SYSTEM DRILL_MVL (* Drill System Model+View+HMI with shared simulation clock *)
  (* Standard: 61499-1; Classification: Simulation; ApplicationDomain: Transfer Lines; Function: Drilling *)
  (* Version 0.1, 2004-10-25, JHC, Rockwell Automation, Adapted to new Load/Unload model. *)
  (* Version 0.0, 2004-09-26, JHC, Rockwell Automation *)
  DEVICE MODEL : FRAME_DEVICE
    RESOURCE CLOCK : EMB_RES
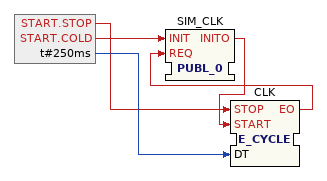
      FBS
        CLK : E_CYCLE;
        SIM_CLK : PUBL_0;
      END_FBS
      EVENT_CONNECTIONS
        START.STOP TO CLK.STOP;
        START.COLD TO SIM_CLK.INIT;
        SIM_CLK.INITO TO CLK.START;
        CLK.EO TO SIM_CLK.REQ;
      END_CONNECTIONS
      DATA_CONNECTIONS
        t#250ms TO CLK.DT;
      END_CONNECTIONS
    END_RESOURCE
    RESOURCE SUPPLY_MDL : EMB_RES
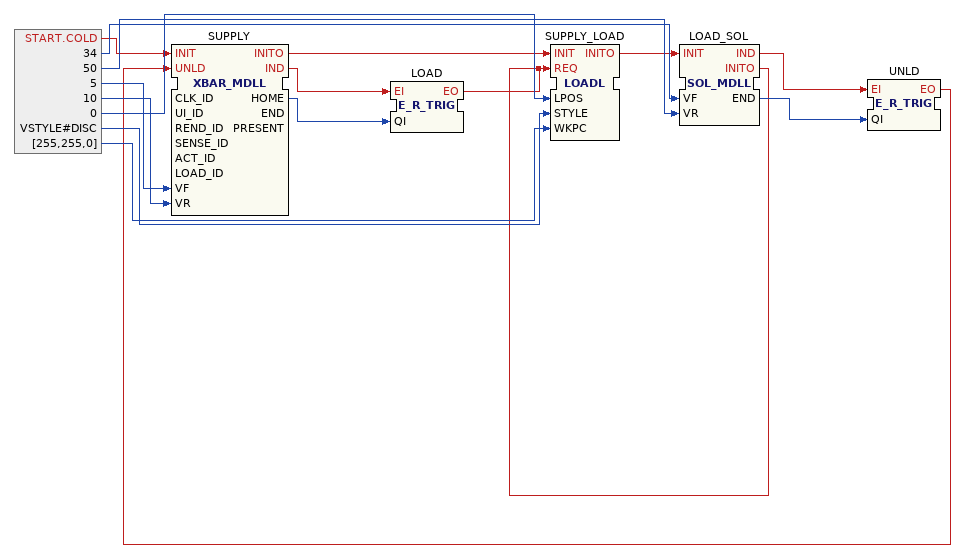
      FBS
        SUPPLY : XBAR_MDLL;
        LOAD_SOL : SOL_MDLL;
        UNLD : E_R_TRIG;
        LOAD : E_R_TRIG;
        SUPPLY_LOAD : LOADL;
      END_FBS
      EVENT_CONNECTIONS
        START.COLD TO SUPPLY.INIT;
        LOAD_SOL.IND TO UNLD.EI;
        SUPPLY.IND TO LOAD.EI;
        UNLD.EO TO SUPPLY.UNLD;
        SUPPLY.INITO TO SUPPLY_LOAD.INIT;
        SUPPLY_LOAD.INITO TO LOAD_SOL.INIT;
        LOAD_SOL.INITO TO SUPPLY_LOAD.REQ;
        LOAD.EO TO SUPPLY_LOAD.REQ;
      END_CONNECTIONS
      DATA_CONNECTIONS
        34 TO LOAD_SOL.VF;
        50 TO LOAD_SOL.VR;
        LOAD_SOL.END TO UNLD.QI;
        5 TO SUPPLY.VF;
        10 TO SUPPLY.VR;
        SUPPLY.HOME TO LOAD.QI;
        0 TO SUPPLY_LOAD.LPOS;
        VSTYLE#DISC TO SUPPLY_LOAD.STYLE;
        [255,255,0] TO SUPPLY_LOAD.WKPC;
      END_CONNECTIONS
    END_RESOURCE
    RESOURCE SLIDE_MDL : EMB_RES
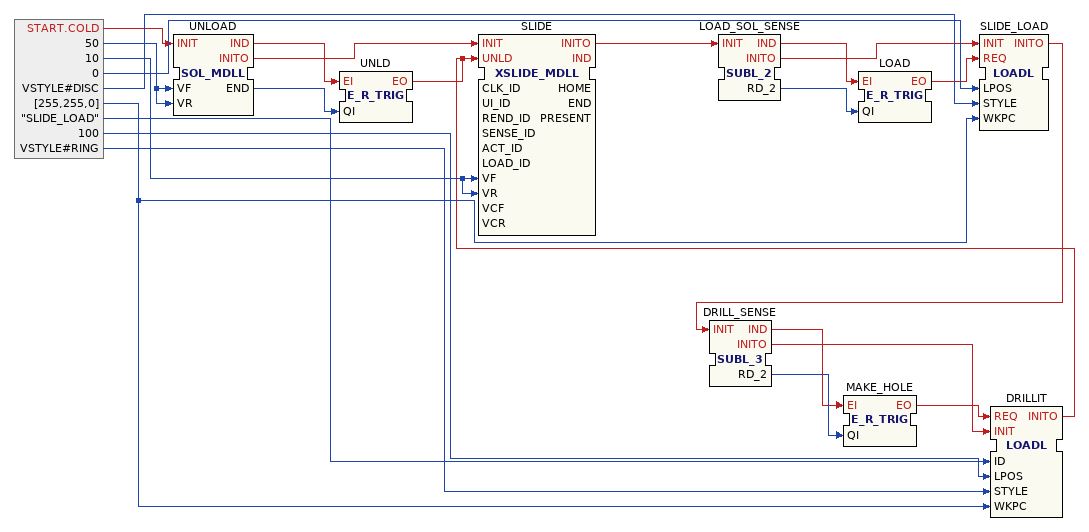
      FBS
        SLIDE : XSLIDE_MDLL;
        UNLOAD : SOL_MDLL;
        DRILL_SENSE : SUBL_3;
        MAKE_HOLE : E_R_TRIG;
        UNLD : E_R_TRIG;
        LOAD_SOL_SENSE : SUBL_2;
        LOAD : E_R_TRIG;
        SLIDE_LOAD : LOADL;
        DRILLIT : LOADL;
      END_FBS
      EVENT_CONNECTIONS
        DRILL_SENSE.IND TO MAKE_HOLE.EI;
        UNLOAD.IND TO UNLD.EI;
        UNLD.EO TO SLIDE.UNLD;
        LOAD_SOL_SENSE.IND TO LOAD.EI;
        START.COLD TO UNLOAD.INIT;
        UNLOAD.INITO TO SLIDE.INIT;
        SLIDE.INITO TO LOAD_SOL_SENSE.INIT;
        LOAD_SOL_SENSE.INITO TO SLIDE_LOAD.INIT;
        LOAD.EO TO SLIDE_LOAD.REQ;
        MAKE_HOLE.EO TO DRILLIT.REQ;
        DRILLIT.INITO TO SLIDE.UNLD;
        SLIDE_LOAD.INITO TO DRILL_SENSE.INIT;
        DRILL_SENSE.INITO TO DRILLIT.INIT;
      END_CONNECTIONS
      DATA_CONNECTIONS
        50 TO UNLOAD.VF;
        50 TO UNLOAD.VR;
        DRILL_SENSE.RD_2 TO MAKE_HOLE.QI;
        10 TO SLIDE.VF;
        10 TO SLIDE.VR;
        UNLOAD.END TO UNLD.QI;
        LOAD_SOL_SENSE.RD_2 TO LOAD.QI;
        0 TO SLIDE_LOAD.LPOS;
        VSTYLE#DISC TO SLIDE_LOAD.STYLE;
        [255,255,0] TO SLIDE_LOAD.WKPC;
        "SLIDE_LOAD" TO DRILLIT.ID;
        100 TO DRILLIT.LPOS;
        VSTYLE#RING TO DRILLIT.STYLE;
        [255,255,0] TO DRILLIT.WKPC;
      END_CONNECTIONS
    END_RESOURCE
    RESOURCE DRILL_MDL : EMB_RES
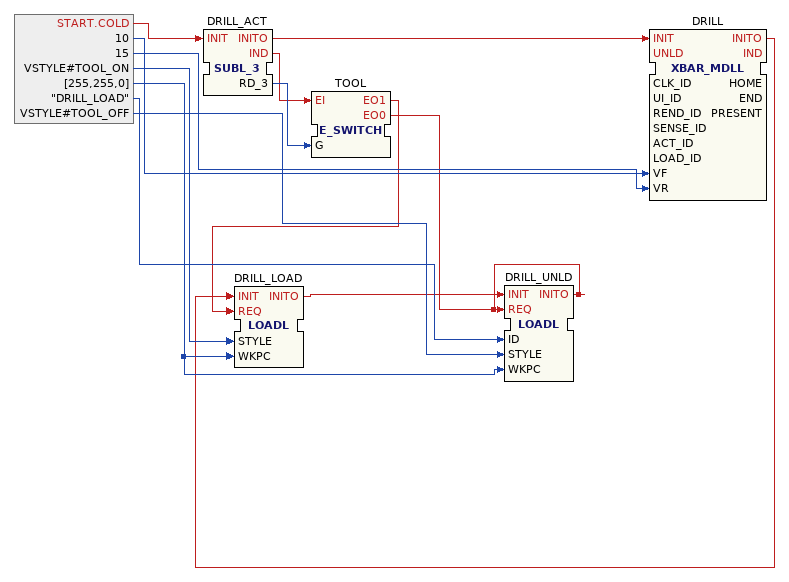
      FBS
        DRILL : XBAR_MDLL;
        DRILL_ACT : SUBL_3;
        TOOL : E_SWITCH;
        DRILL_LOAD : LOADL;
        DRILL_UNLD : LOADL;
      END_FBS
      EVENT_CONNECTIONS
        START.COLD TO DRILL_ACT.INIT;
        DRILL_ACT.INITO TO DRILL.INIT;
        DRILL.INITO TO DRILL_LOAD.INIT;
        DRILL_LOAD.INITO TO DRILL_UNLD.INIT;
        DRILL_ACT.IND TO TOOL.EI;
        TOOL.EO1 TO DRILL_LOAD.REQ;
        TOOL.EO0 TO DRILL_UNLD.REQ;
        DRILL_UNLD.INITO TO DRILL_UNLD.REQ;
      END_CONNECTIONS
      DATA_CONNECTIONS
        10 TO DRILL.VF;
        15 TO DRILL.VR;
        VSTYLE#TOOL_ON TO DRILL_LOAD.STYLE;
        [255,255,0] TO DRILL_LOAD.WKPC;
        "DRILL_LOAD" TO DRILL_UNLD.ID;
        VSTYLE#TOOL_OFF TO DRILL_UNLD.STYLE;
        [255,255,0] TO DRILL_UNLD.WKPC;
        DRILL_ACT.RD_3 TO TOOL.G;
      END_CONNECTIONS
    END_RESOURCE
    RESOURCE TAKEOFF_MDL : EMB_RES
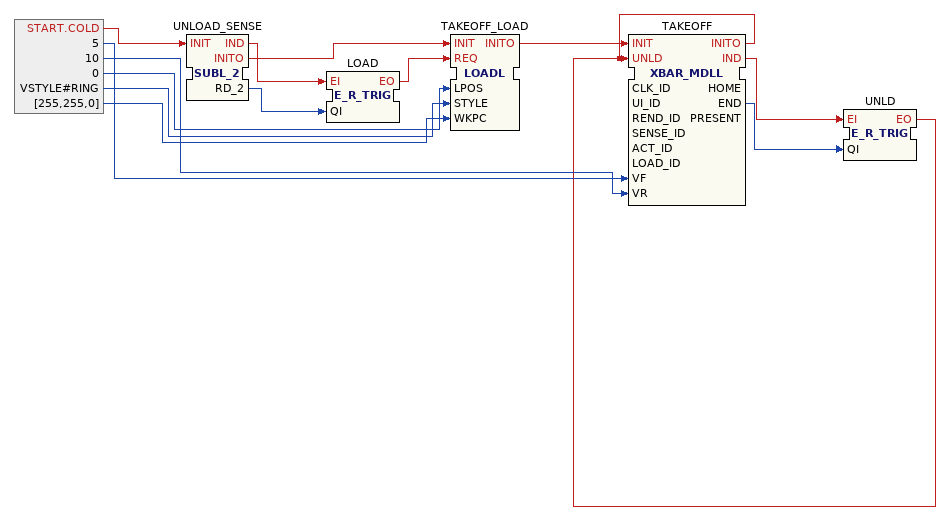
      FBS
        UNLOAD_SENSE : SUBL_2;
        TAKEOFF : XBAR_MDLL;
        UNLD : E_R_TRIG;
        LOAD : E_R_TRIG;
        TAKEOFF_LOAD : LOADL;
      END_FBS
      EVENT_CONNECTIONS
        START.COLD TO UNLOAD_SENSE.INIT;
        UNLD.EO TO TAKEOFF.UNLD;
        TAKEOFF.IND TO UNLD.EI;
        TAKEOFF.INITO TO TAKEOFF.UNLD;
        UNLOAD_SENSE.IND TO LOAD.EI;
        UNLOAD_SENSE.INITO TO TAKEOFF_LOAD.INIT;
        TAKEOFF_LOAD.INITO TO TAKEOFF.INIT;
        LOAD.EO TO TAKEOFF_LOAD.REQ;
      END_CONNECTIONS
      DATA_CONNECTIONS
        TAKEOFF.END TO UNLD.QI;
        5 TO TAKEOFF.VF;
        10 TO TAKEOFF.VR;
        UNLOAD_SENSE.RD_2 TO LOAD.QI;
        0 TO TAKEOFF_LOAD.LPOS;
        VSTYLE#RING TO TAKEOFF_LOAD.STYLE;
        [255,255,0] TO TAKEOFF_LOAD.WKPC;
      END_CONNECTIONS
    END_RESOURCE
    RESOURCE INPUT_VIEW : VIEW_PANEL
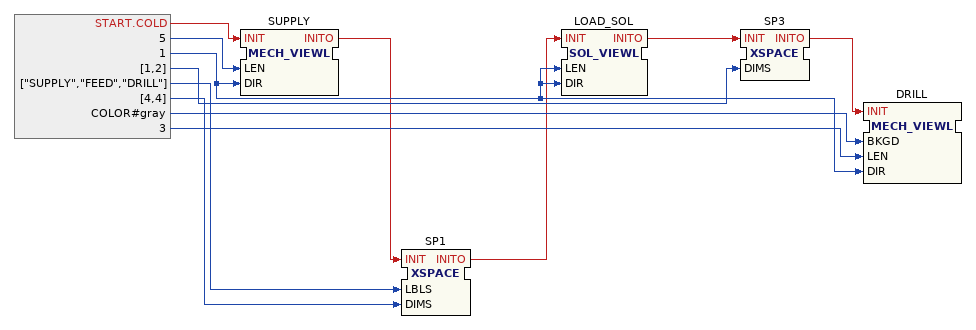
      FBS
        SUPPLY : MECH_VIEWL; (* Supply transfer mechanism *)
        SP1 : XSPACE;
        LOAD_SOL : SOL_VIEWL; (* Loader mechanism *)
        SP3 : XSPACE;
        DRILL : MECH_VIEWL;
      END_FBS
      EVENT_CONNECTIONS
        START.COLD TO SUPPLY.INIT;
        SUPPLY.INITO TO SP1.INIT;
        SP1.INITO TO LOAD_SOL.INIT;
        LOAD_SOL.INITO TO SP3.INIT;
        SP3.INITO TO DRILL.INIT;
      END_CONNECTIONS
      DATA_CONNECTIONS
        5 TO SUPPLY.LEN;
        1 TO SUPPLY.DIR;
        [1,2] TO SP3.DIMS;
        ["SUPPLY","FEED","DRILL"] TO SP1.LBLS;
        [4,4] TO SP1.DIMS;
        COLOR#gray TO DRILL.BKGD;
        3 TO DRILL.LEN;
        1 TO DRILL.DIR;
        1 TO LOAD_SOL.LEN;
        1 TO LOAD_SOL.DIR;
      END_CONNECTIONS
    END_RESOURCE
    RESOURCE OUTPUT_VIEW : VIEW_PANEL
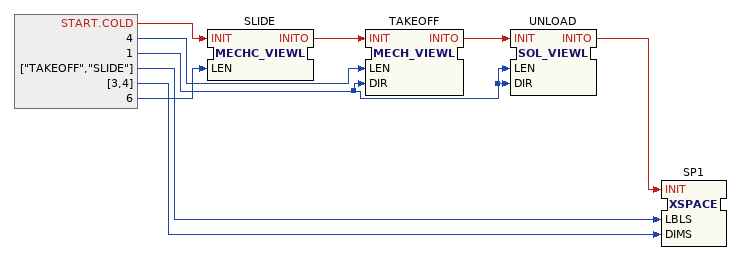
      FBS
        SLIDE : MECHC_VIEWL;
        TAKEOFF : MECH_VIEWL; (* Takeoff Transfer *)
        UNLOAD : SOL_VIEWL; (* Unloader Mechanism *)
        SP1 : XSPACE;
      END_FBS
      EVENT_CONNECTIONS
        START.COLD TO SLIDE.INIT;
        SLIDE.INITO TO TAKEOFF.INIT;
        TAKEOFF.INITO TO UNLOAD.INIT;
        UNLOAD.INITO TO SP1.INIT;
      END_CONNECTIONS
      DATA_CONNECTIONS
        4 TO TAKEOFF.LEN;
        1 TO TAKEOFF.DIR;
        ["TAKEOFF","SLIDE"] TO SP1.LBLS;
        [3,4] TO SP1.DIMS;
        1 TO UNLOAD.LEN;
        1 TO UNLOAD.DIR;
        6 TO SLIDE.LEN;
      END_CONNECTIONS
    END_RESOURCE
    DATA_CONNECTIONS
      0 TO INPUT_VIEW.TRACE;
      30 TO INPUT_VIEW.DIA;
      [6,5] TO INPUT_VIEW.SIZE;
      1 TO INPUT_VIEW.VERTICAL;
      30 TO OUTPUT_VIEW.DIA;
      [6,5] TO OUTPUT_VIEW.SIZE;
    END_CONNECTIONS
  END_DEVICE
  DEVICE HMI : FRAME_DEVICE
    RESOURCE SUPPLY_SENSORS : PANEL_RESOURCE
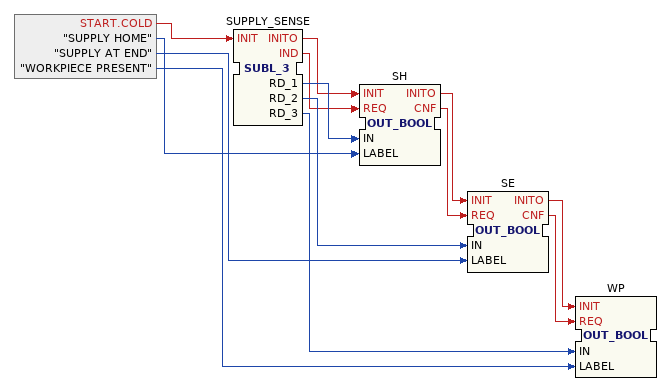
      FBS
        SUPPLY_SENSE : SUBL_3;
        SH : OUT_BOOL;
        SE : OUT_BOOL;
        WP : OUT_BOOL;
      END_FBS
      EVENT_CONNECTIONS
        START.COLD TO SUPPLY_SENSE.INIT;
        SUPPLY_SENSE.INITO TO SH.INIT;
        SH.INITO TO SE.INIT;
        SE.INITO TO WP.INIT;
        SUPPLY_SENSE.IND TO SH.REQ;
        SH.CNF TO SE.REQ;
        SE.CNF TO WP.REQ;
      END_CONNECTIONS
      DATA_CONNECTIONS
        SUPPLY_SENSE.RD_1 TO SH.IN;
        SUPPLY_SENSE.RD_2 TO SE.IN;
        SUPPLY_SENSE.RD_3 TO WP.IN;
        "SUPPLY HOME" TO SH.LABEL;
        "SUPPLY AT END" TO SE.LABEL;
        "WORKPIECE PRESENT" TO WP.LABEL;
      END_CONNECTIONS
    END_RESOURCE
    RESOURCE SUPPLY_ACTUATORS : PANEL_RESOURCE
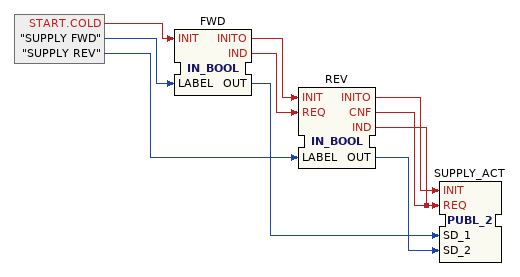
      FBS
        FWD : IN_BOOL;
        REV : IN_BOOL;
        SUPPLY_ACT : PUBL_2;
      END_FBS
      EVENT_CONNECTIONS
        START.COLD TO FWD.INIT;
        FWD.INITO TO REV.INIT;
        REV.INITO TO SUPPLY_ACT.INIT;
        FWD.IND TO REV.REQ;
        REV.CNF TO SUPPLY_ACT.REQ;
        REV.IND TO SUPPLY_ACT.REQ;
      END_CONNECTIONS
      DATA_CONNECTIONS
        FWD.OUT TO SUPPLY_ACT.SD_1;
        REV.OUT TO SUPPLY_ACT.SD_2;
        "SUPPLY FWD" TO FWD.LABEL;
        "SUPPLY REV" TO REV.LABEL;
      END_CONNECTIONS
    END_RESOURCE
    RESOURCE LOAD_SENSORS : PANEL_RESOURCE
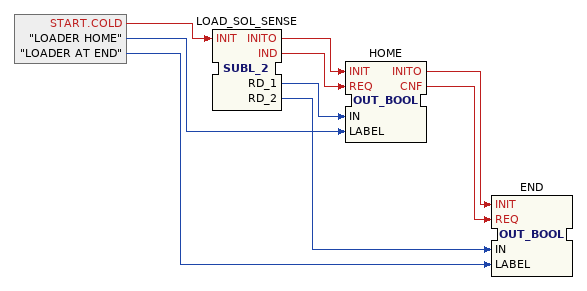
      FBS
        LOAD_SOL_SENSE : SUBL_2;
        HOME : OUT_BOOL;
        END : OUT_BOOL;
      END_FBS
      EVENT_CONNECTIONS
        START.COLD TO LOAD_SOL_SENSE.INIT;
        LOAD_SOL_SENSE.INITO TO HOME.INIT;
        HOME.INITO TO END.INIT;
        LOAD_SOL_SENSE.IND TO HOME.REQ;
        HOME.CNF TO END.REQ;
      END_CONNECTIONS
      DATA_CONNECTIONS
        LOAD_SOL_SENSE.RD_1 TO HOME.IN;
        LOAD_SOL_SENSE.RD_2 TO END.IN;
        "LOADER HOME" TO HOME.LABEL;
        "LOADER AT END" TO END.LABEL;
      END_CONNECTIONS
    END_RESOURCE
    RESOURCE LOAD_ACTUATORS : PANEL_RESOURCE
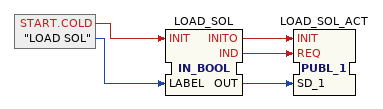
      FBS
        LOAD_SOL : IN_BOOL;
        LOAD_SOL_ACT : PUBL_1;
      END_FBS
      EVENT_CONNECTIONS
        START.COLD TO LOAD_SOL.INIT;
        LOAD_SOL.INITO TO LOAD_SOL_ACT.INIT;
        LOAD_SOL.IND TO LOAD_SOL_ACT.REQ;
      END_CONNECTIONS
      DATA_CONNECTIONS
        LOAD_SOL.OUT TO LOAD_SOL_ACT.SD_1;
        "LOAD SOL" TO LOAD_SOL.LABEL;
      END_CONNECTIONS
    END_RESOURCE
    RESOURCE SLIDE_SENSORS : PANEL_RESOURCE
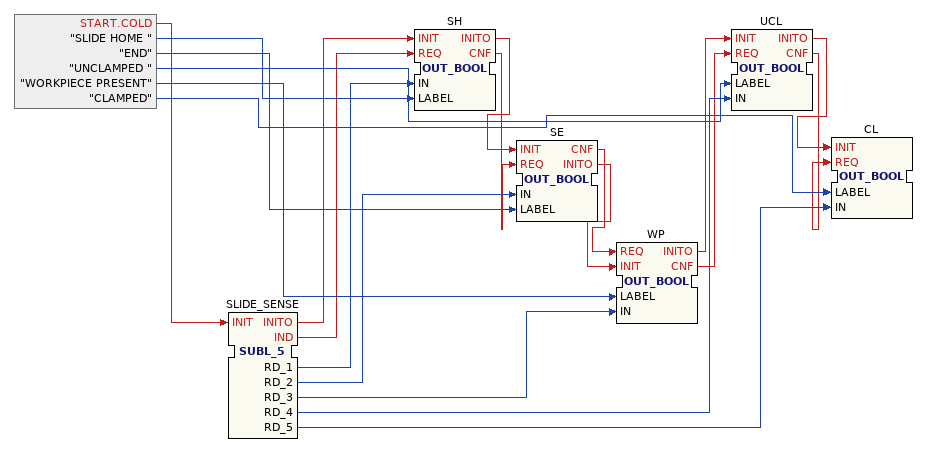
      FBS
        SLIDE_SENSE : SUBL_5;
        SH : OUT_BOOL;
        SE : OUT_BOOL;
        UCL : OUT_BOOL;
        CL : OUT_BOOL;
        WP : OUT_BOOL;
      END_FBS
      EVENT_CONNECTIONS
        START.COLD TO SLIDE_SENSE.INIT;
        SLIDE_SENSE.INITO TO SH.INIT;
        SH.INITO TO SE.INIT;
        UCL.INITO TO CL.INIT;
        SLIDE_SENSE.IND TO SH.REQ;
        SH.CNF TO SE.REQ;
        UCL.CNF TO CL.REQ;
        SE.CNF TO WP.REQ;
        SE.INITO TO WP.INIT;
        WP.INITO TO UCL.INIT;
        WP.CNF TO UCL.REQ;
      END_CONNECTIONS
      DATA_CONNECTIONS
        SLIDE_SENSE.RD_1 TO SH.IN;
        SLIDE_SENSE.RD_2 TO SE.IN;
        "SLIDE HOME " TO SH.LABEL;
        "END" TO SE.LABEL;
        "UNCLAMPED " TO UCL.LABEL;
        "WORKPIECE PRESENT" TO WP.LABEL;
        "CLAMPED" TO CL.LABEL;
        SLIDE_SENSE.RD_3 TO WP.IN;
        SLIDE_SENSE.RD_4 TO UCL.IN;
        SLIDE_SENSE.RD_5 TO CL.IN;
      END_CONNECTIONS
    END_RESOURCE
    RESOURCE SLIDE_ACTUATORS : PANEL_RESOURCE
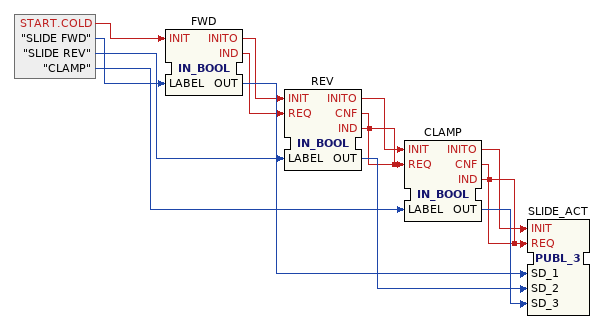
      FBS
        FWD : IN_BOOL;
        REV : IN_BOOL;
        CLAMP : IN_BOOL;
        SLIDE_ACT : PUBL_3;
      END_FBS
      EVENT_CONNECTIONS
        START.COLD TO FWD.INIT;
        FWD.INITO TO REV.INIT;
        REV.INITO TO CLAMP.INIT;
        CLAMP.INITO TO SLIDE_ACT.INIT;
        FWD.IND TO REV.REQ;
        REV.CNF TO CLAMP.REQ;
        REV.IND TO CLAMP.REQ;
        CLAMP.CNF TO SLIDE_ACT.REQ;
        CLAMP.IND TO SLIDE_ACT.REQ;
      END_CONNECTIONS
      DATA_CONNECTIONS
        FWD.OUT TO SLIDE_ACT.SD_1;
        REV.OUT TO SLIDE_ACT.SD_2;
        CLAMP.OUT TO SLIDE_ACT.SD_3;
        "SLIDE FWD" TO FWD.LABEL;
        "SLIDE REV" TO REV.LABEL;
        "CLAMP" TO CLAMP.LABEL;
      END_CONNECTIONS
    END_RESOURCE
    RESOURCE DRILL_SENSORS : PANEL_RESOURCE
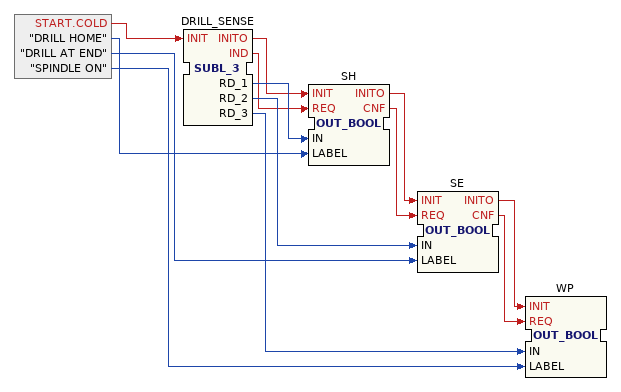
      FBS
        DRILL_SENSE : SUBL_3;
        SH : OUT_BOOL;
        SE : OUT_BOOL;
        WP : OUT_BOOL;
      END_FBS
      EVENT_CONNECTIONS
        START.COLD TO DRILL_SENSE.INIT;
        DRILL_SENSE.INITO TO SH.INIT;
        SH.INITO TO SE.INIT;
        SE.INITO TO WP.INIT;
        DRILL_SENSE.IND TO SH.REQ;
        SH.CNF TO SE.REQ;
        SE.CNF TO WP.REQ;
      END_CONNECTIONS
      DATA_CONNECTIONS
        DRILL_SENSE.RD_1 TO SH.IN;
        DRILL_SENSE.RD_2 TO SE.IN;
        DRILL_SENSE.RD_3 TO WP.IN;
        "DRILL HOME" TO SH.LABEL;
        "DRILL AT END" TO SE.LABEL;
        "SPINDLE ON" TO WP.LABEL;
      END_CONNECTIONS
    END_RESOURCE
    RESOURCE DRILL_ACTUATORS : PANEL_RESOURCE
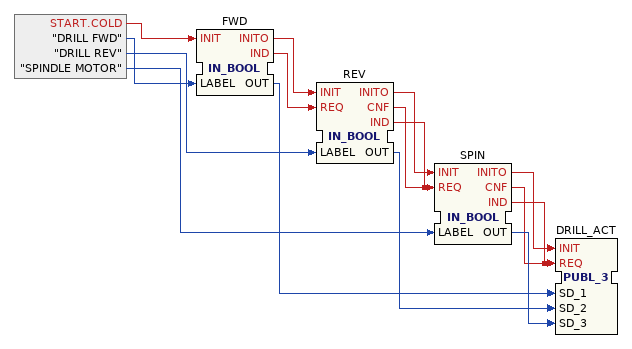
      FBS
        FWD : IN_BOOL;
        REV : IN_BOOL;
        SPIN : IN_BOOL;
        DRILL_ACT : PUBL_3;
      END_FBS
      EVENT_CONNECTIONS
        START.COLD TO FWD.INIT;
        FWD.INITO TO REV.INIT;
        REV.INITO TO SPIN.INIT;
        SPIN.INITO TO DRILL_ACT.INIT;
        FWD.IND TO REV.REQ;
        REV.CNF TO SPIN.REQ;
        REV.IND TO SPIN.REQ;
        SPIN.CNF TO DRILL_ACT.REQ;
        SPIN.IND TO DRILL_ACT.REQ;
      END_CONNECTIONS
      DATA_CONNECTIONS
        FWD.OUT TO DRILL_ACT.SD_1;
        REV.OUT TO DRILL_ACT.SD_2;
        SPIN.OUT TO DRILL_ACT.SD_3;
        "DRILL FWD" TO FWD.LABEL;
        "DRILL REV" TO REV.LABEL;
        "SPINDLE MOTOR" TO SPIN.LABEL;
      END_CONNECTIONS
    END_RESOURCE
    RESOURCE UNLOAD_SENSORS : PANEL_RESOURCE
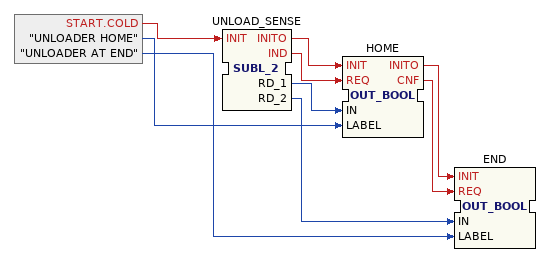
      FBS
        UNLOAD_SENSE : SUBL_2;
        HOME : OUT_BOOL;
        END : OUT_BOOL;
      END_FBS
      EVENT_CONNECTIONS
        START.COLD TO UNLOAD_SENSE.INIT;
        UNLOAD_SENSE.INITO TO HOME.INIT;
        HOME.INITO TO END.INIT;
        UNLOAD_SENSE.IND TO HOME.REQ;
        HOME.CNF TO END.REQ;
      END_CONNECTIONS
      DATA_CONNECTIONS
        UNLOAD_SENSE.RD_1 TO HOME.IN;
        UNLOAD_SENSE.RD_2 TO END.IN;
        "UNLOADER HOME" TO HOME.LABEL;
        "UNLOADER AT END" TO END.LABEL;
      END_CONNECTIONS
    END_RESOURCE
    RESOURCE UNLOAD_ACTUATORS : PANEL_RESOURCE
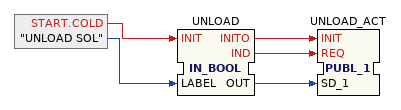
      FBS
        UNLOAD : IN_BOOL;
        UNLOAD_ACT : PUBL_1;
      END_FBS
      EVENT_CONNECTIONS
        START.COLD TO UNLOAD.INIT;
        UNLOAD.INITO TO UNLOAD_ACT.INIT;
        UNLOAD.IND TO UNLOAD_ACT.REQ;
      END_CONNECTIONS
      DATA_CONNECTIONS
        UNLOAD.OUT TO UNLOAD_ACT.SD_1;
        "UNLOAD SOL" TO UNLOAD.LABEL;
      END_CONNECTIONS
    END_RESOURCE
    RESOURCE TAKEOFF_SENSORS : PANEL_RESOURCE
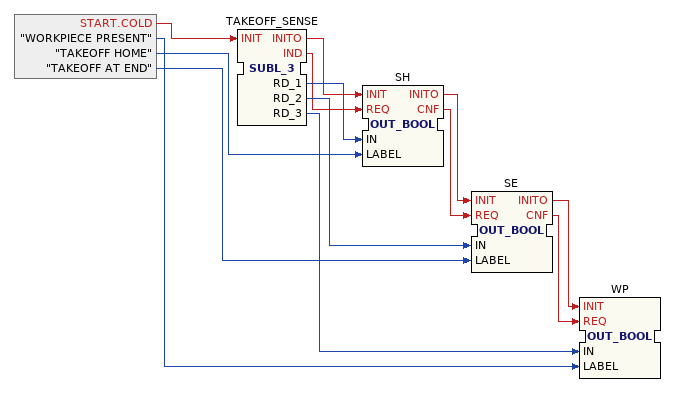
      FBS
        TAKEOFF_SENSE : SUBL_3;
        SH : OUT_BOOL;
        SE : OUT_BOOL;
        WP : OUT_BOOL;
      END_FBS
      EVENT_CONNECTIONS
        START.COLD TO TAKEOFF_SENSE.INIT;
        TAKEOFF_SENSE.INITO TO SH.INIT;
        SH.INITO TO SE.INIT;
        SE.INITO TO WP.INIT;
        TAKEOFF_SENSE.IND TO SH.REQ;
        SH.CNF TO SE.REQ;
        SE.CNF TO WP.REQ;
      END_CONNECTIONS
      DATA_CONNECTIONS
        TAKEOFF_SENSE.RD_1 TO SH.IN;
        TAKEOFF_SENSE.RD_2 TO SE.IN;
        TAKEOFF_SENSE.RD_3 TO WP.IN;
        "WORKPIECE PRESENT" TO WP.LABEL;
        "TAKEOFF HOME" TO SH.LABEL;
        "TAKEOFF AT END" TO SE.LABEL;
      END_CONNECTIONS
    END_RESOURCE
    RESOURCE TAKEOFF_ACTUATORS : PANEL_RESOURCE
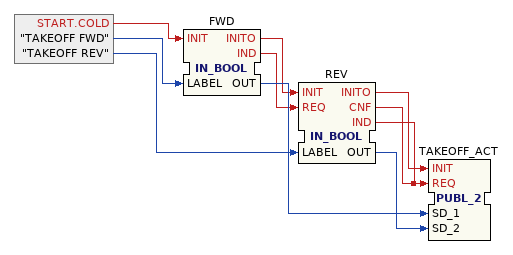
      FBS
        FWD : IN_BOOL;
        REV : IN_BOOL;
        TAKEOFF_ACT : PUBL_2;
      END_FBS
      EVENT_CONNECTIONS
        START.COLD TO FWD.INIT;
        FWD.INITO TO REV.INIT;
        REV.INITO TO TAKEOFF_ACT.INIT;
        FWD.IND TO REV.REQ;
        REV.CNF TO TAKEOFF_ACT.REQ;
        REV.IND TO TAKEOFF_ACT.REQ;
      END_CONNECTIONS
      DATA_CONNECTIONS
        FWD.OUT TO TAKEOFF_ACT.SD_1;
        REV.OUT TO TAKEOFF_ACT.SD_2;
        "TAKEOFF FWD" TO FWD.LABEL;
        "TAKEOFF REV" TO REV.LABEL;
      END_CONNECTIONS
    END_RESOURCE
  END_DEVICE
  DATA_CONNECTIONS (* parameter values *)
    [100,100,375,360] TO HMI.BOUNDS;
    [6,2] TO HMI.GRID;
    [475,100,190,360] TO MODEL.BOUNDS;
  END_CONNECTIONS
END_SYSTEM
